Xinje XDPPro project, PLC1: XDH-60T4 (software 3.7.14b 2022-06-24)

PROGRAM 梯形图

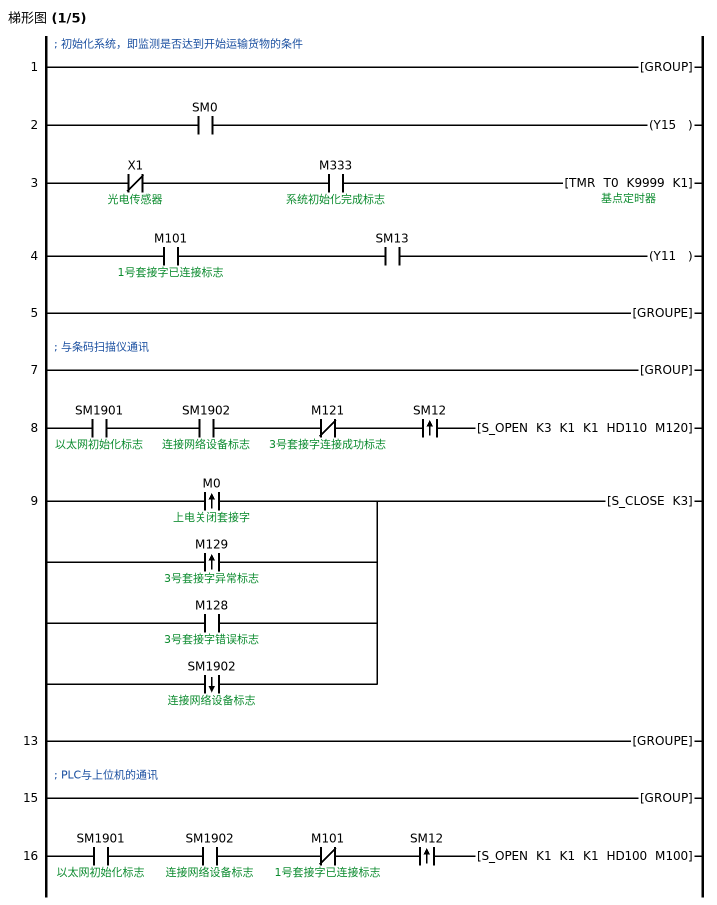
; 初始化系统，即监测是否达到开始运输货物的条件
GROUP
LD     SM0
OUT    Y15
LDI    X1	; 光电传感器
AND    M333	; 系统初始化完成标志
TMR    T0 K9999 K1	; 基点定时器
LD     M101	; 1号套接字已连接标志
AND    SM13
OUT    Y11
GROUPE
; 与条码扫描仪通讯
GROUP
LD     SM1901	; 以太网初始化标志
AND    SM1902	; 连接网络设备标志
ANI    M121	; 3号套接字连接成功标志
ANDP   SM12
S_OPEN K3 K1 K1 HD110 M120
LDP    M0	; 上电关闭套接字
ORP    M129	; 3号套接字异常标志
OR     M128	; 3号套接字错误标志
ORF    SM1902	; 连接网络设备标志
S_CLOSE K3
GROUPE
; PLC与上位机的通讯
GROUP
LD     SM1901	; 以太网初始化标志
AND    SM1902	; 连接网络设备标志
ANI    M101	; 1号套接字已连接标志
ANDP   SM12
S_OPEN K1 K1 K1 HD100 M100

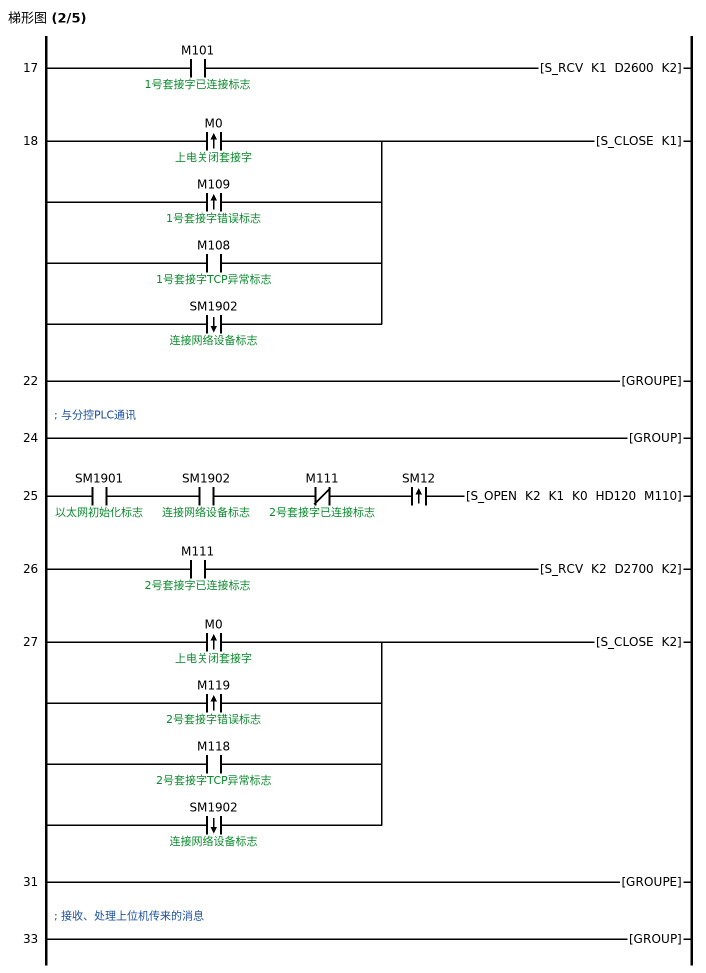
LD     M101	; 1号套接字已连接标志
S_RCV  K1 D2600 K2
LDP    M0	; 上电关闭套接字
ORP    M109	; 1号套接字错误标志
OR     M108	; 1号套接字TCP异常标志
ORF    SM1902	; 连接网络设备标志
S_CLOSE K1
GROUPE
; 与分控PLC通讯
GROUP
LD     SM1901	; 以太网初始化标志
AND    SM1902	; 连接网络设备标志
ANI    M111	; 2号套接字已连接标志
ANDP   SM12
S_OPEN K2 K1 K0 HD120 M110
LD     M111	; 2号套接字已连接标志
S_RCV  K2 D2700 K2
LDP    M0	; 上电关闭套接字
ORP    M119	; 2号套接字错误标志
OR     M118	; 2号套接字TCP异常标志
ORF    SM1902	; 连接网络设备标志
S_CLOSE K2
GROUPE
; 接收、处理上位机传来的消息
GROUP

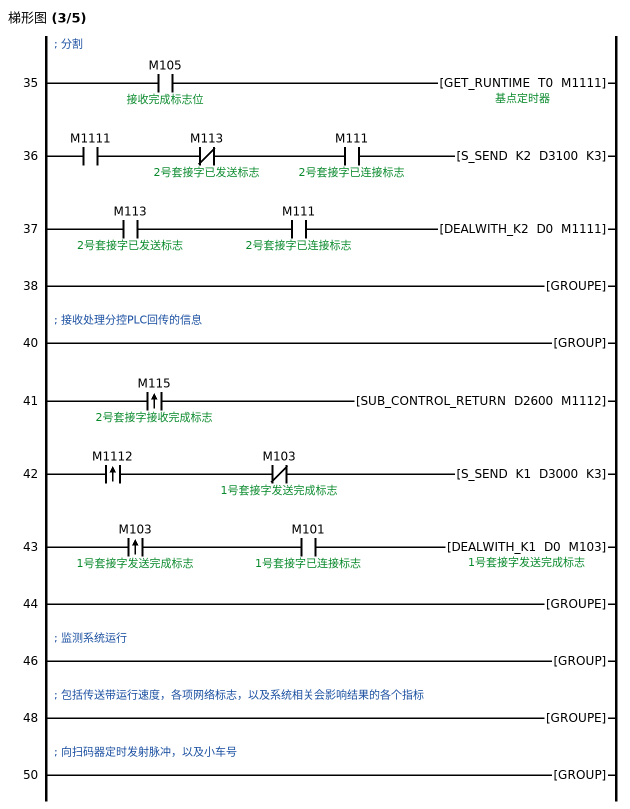
; 分割
LD     M105	; 接收完成标志位
GET_RUNTIME T0 M1111	; 基点定时器
LD     M1111
ANI    M113	; 2号套接字已发送标志
AND    M111	; 2号套接字已连接标志
S_SEND K2 D3100 K3
LD     M113	; 2号套接字已发送标志
AND    M111	; 2号套接字已连接标志
DEALWITH_K2 D0 M1111
GROUPE
; 接收处理分控PLC回传的信息
GROUP
LDP    M115	; 2号套接字接收完成标志
SUB_CONTROL_RETURN D2600 M1112
LDP    M1112
ANI    M103	; 1号套接字发送完成标志
S_SEND K1 D3000 K3
LDP    M103	; 1号套接字发送完成标志
AND    M101	; 1号套接字已连接标志
DEALWITH_K1 D0 M103	; 1号套接字发送完成标志
GROUPE
; 监测系统运行
GROUP
; 包括传送带运行速度，各项网络标志，以及系统相关会影响结果的各个指标
GROUPE
; 向扫码器定时发射脉冲，以及小车号
GROUP

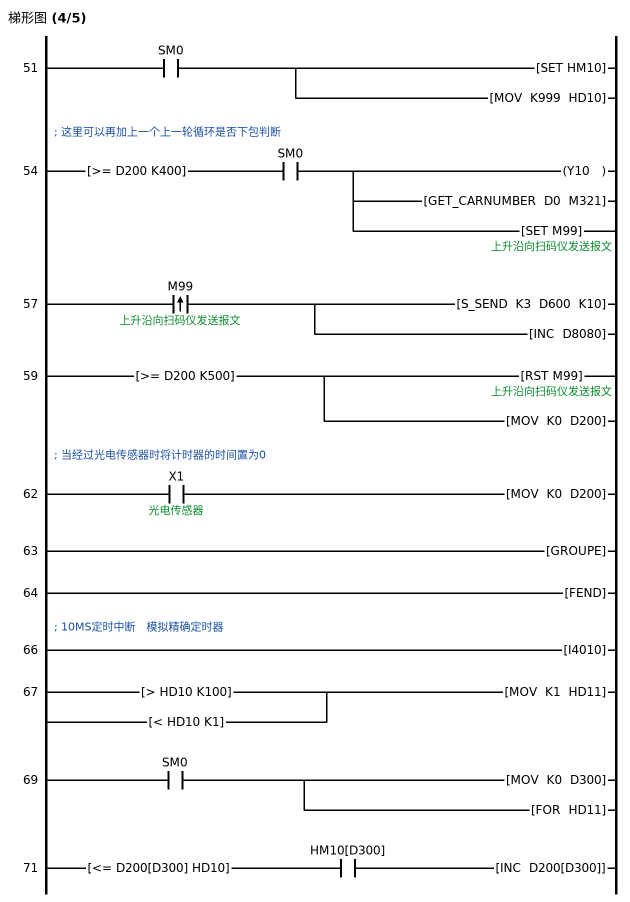
LD     SM0
SET    HM10
MOV    K999 HD10
; 这里可以再加上一个上一轮循环是否下包判断
LD>=   D200 K400
AND    SM0
OUT    Y10
GET_CARNUMBER D0 M321
SET    M99	; 上升沿向扫码仪发送报文
LDP    M99	; 上升沿向扫码仪发送报文
S_SEND K3 D600 K10
INC    D8080
LD>=   D200 K500
RST    M99	; 上升沿向扫码仪发送报文
MOV    K0 D200
; 当经过光电传感器时将计时器的时间置为0
LD     X1	; 光电传感器
MOV    K0 D200
GROUPE
FEND
; 10MS定时中断　模拟精确定时器
I4010
LD>    HD10 K100
OR<    HD10 K1
MOV    K1 HD11
LD     SM0
MOV    K0 D300
FOR    HD11
LD<=   D200[D300] HD10
AND    HM10[D300]
INC    D200[D300]

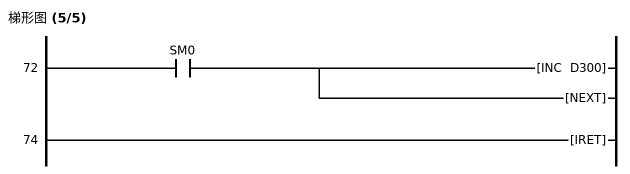
LD     SM0
INC    D300
NEXT
IRET

COMMENTS (devices not used above)
M1	1号套接字发送数据标志
HM0	手动建立连接
M2	1号套接字接收数据
M3	2号套接字发送数据标志
M4	2号套接字接收数据标志
Y6	给相机发脉冲
Y0	相机
Y7	接扫码仪

C FILE func1.h
#ifndef	_FUNC1_H
#define	_FUNC1_H
/*********宏定义用来存放需要的返回值************/
 #define NEEDTIME D[3100]       //保存返回值
 #define CAR      D[2600]        //存储判断出来的小车号
 #define Bourn     D[2605]       //目的格口
//#define Time      D[300]           //时间基点定时器的计数值 
#define D_D	     *(INT32S*)&D

/* 存放一些函数中需要的参数 
所有的距离单位为毫米，时间单位为毫秒
 */
 #define tmpp D_D[798]
 #define carnumber D_D[598]
 
 
INT32S TrackLength = 50000;           //轨道的长度
INT32S  Speed = 1;               //小车速度1mm/ms
INT32S DistanceOfCar = 400;      //小车的间距(单位为：毫米)
INT32S TIMELOSS = 5;          //电机启动时间偏移量(单位为：毫秒)

INT32S Time_Offset =0 ;           //时间偏移量，由于没有进行实验测试暂时设置为0,该值是用来计算小车上的电机转动所需要的时间

INT32S DistanceOfCut = 900;          //此处割口的间距 ————割口的长度加上割口间的距离

INT32S  Camera_Position = 600; //扫码设备的位置

INT32S Time = 0;               //距离时间基点的时间

INT32S Failure[20];

#endif

C FUNCTION BLOCK dealwith_k1.fcb
/* #EXPORT_ENTRY_BEGIN(DEALWITH_K1)
//    类型              模式             个数               映射          注释
W = { type = "PINT16S", mode = [In,Out], count = "unknown", map = [D,HD], comment = "" }
B = { type = "BIT"    , mode = [In,Out], count = "unknown", map = [M,HM], comment = "" }
#EXPORT_ENTRY_END */
/*************************************************************************
 * FunctionBlockName:  DEALWITH_K1
 * Version:            1.0.0
 * Author:             
 * UpdateTime:         2022-08-22 14:10:12
 * Comment:            
**************************************************************************/

/**
 * @summary 
 * @param W 
 * @param B 
 */
void DEALWITH_K1(PINT16S W,BIT B)
{
	#define SysRegAddr_HD_D_HM_M
    M[103] = 0;

}

C FUNCTION BLOCK dealwith_k2.fcb
/* #EXPORT_ENTRY_BEGIN(DEALWITH_K2)
//    类型              模式             个数               映射          注释
W = { type = "PINT16S", mode = [In,Out], count = "unknown", map = [D,HD], comment = "" }
B = { type = "BIT"    , mode = [In,Out], count = "unknown", map = [M,HM], comment = "" }
#EXPORT_ENTRY_END */
/*************************************************************************
 * FunctionBlockName:  DEALWITH_K2
 * Version:            1.0.0
 * Author:             
 * UpdateTime:         2022-08-22 14:08:06
 * Comment:            
**************************************************************************/

/**
 * @summary 
 * @param W 
 * @param B 
 */
void DEALWITH_K2(PINT16S W,BIT B)
{
	#define SysRegAddr_HD_D_HM_M
    M[113] = 0;
    M[1111] = 0;

}

C FUNCTION BLOCK func1.fcb
/* #EXPORT_ENTRY_BEGIN(FUNC1)
//    类型              模式             个数               映射          注释
W = { type = "PINT16S", mode = [In,Out], count = "unknown", map = [D,HD], comment = "" }
B = { type = "BIT"    , mode = [In,Out], count = "unknown", map = [M,HM], comment = "" }
#EXPORT_ENTRY_END */
/*************************************************************************
 * FunctionBlockName:  FUNC1
 * Version:            1.0.0
 * Author:             
 * UpdateTime:         2022-08-18 08:24:01
 * Comment:            
**************************************************************************/

/**
 * @summary 
 * @param W 
 * @param B 
 */
void FUNC1(PINT16S W,BIT B)
{
	#define SysRegAddr_HD_D_HM_M

}

C FUNCTION BLOCK get_carnumber.fcb
/* 输入时间，返回当前相机拍摄的小车号
#EXPORT_ENTRY_BEGIN(GET_CARNUMBER)
//    类型              模式             个数               映射          注释
W = { type = "PINT16S", mode = [In,Out], count = "unknown", map = [D,HD], comment = "" }
B = { type = "BIT"    , mode = [In,Out], count = "unknown", map = [M,HM], comment = "" }
#EXPORT_ENTRY_END */
/*************************************************************************
 * FunctionBlockName:  GET_CARNUMBER
 * Version:            1.0.0
 * Author:             rpl
 * UpdateTime:         2022-08-10 14:44:36
 * Comment:            输入时间，返回当前相机拍摄的小车号
**************************************************************************/

/**
 * @summary 
 * @param W 
 * @param B 
 */
 #include"func1.h"
 
 
void GET_CARNUMBER(PINT16S W,BIT B)
{
	#define SysRegAddr_HD_D_HM_M＿T
	/*根据时间判断出当前是多少号小车(小车从0号开始排序) */
     tmpp =  Speed * D[888] *10- Camera_Position;
    carnumber = ( tmpp / DistanceOfCar );  //判断是哪个小车，用来绑定小车的控制电机计时时间
    //CAR = 40;
    /***判断小车上的货物是否在上一轮没有卸载下来,暂不判断******/ 

    
    /***将小车号数据写入寄存器，起始位置Ｄ600,十个***/
        //消息头
    D[600] = 0x02;
    //功能位
    D[601] = 0x53;
    //千位
    D[602] = 0x30;
    
    //百位
    int ss= (D[598] /100) % 10；
    D[603] = 48+ss;
    
    //十位
    int  temp = 48 + (D[598] /10) % 10；
    D[604] = temp;
    
    //个位
    int  temp0 = 48 + D[598] % 10；
    D[605] = temp0;
    
    //结束符
    D[606] = 0x03;
    unsigned char LRC = 0;
    for(int i = 601;i<=605;i++)
    {
        LRC ^= D[i];
    }
    //LRC 校验
    D[607] = LRC;
    
    //尾字符
    D[608] = 0x0D;
    D[609] = 0x0A;
    
    
    
    M[321] = 1;
    return;
}

C FUNCTION BLOCK get_runtime.fcb
/* D[100]返回某个电机在多少秒后运行,D[101]返回判断出的小车号，以此来进行绑定
#EXPORT_ENTRY_BEGIN(GET_RUNTIME)
//    类型          模式             个数               映射          注释
w = { type = "BIT", mode = [In]    , count = "1"      , map = [T]   , comment = "时间差" }
B = { type = "BIT", mode = [In,Out], count = "unknown", map = [M,HM], comment = ""    }
#EXPORT_ENTRY_END */
/*************************************************************************
 * FunctionBlockName:  GET_RUNTIME
 * Version:            1.0.0
 * Author:             rpl
 * UpdateTime:         2022-07-25 16:38:06
 * Comment:            D[100]返回某个电机在多少秒后运行,D[101]返回判断出的小车号，以此来进行绑定
**************************************************************************/

/**
 * @summary 
 * @param w 时间差
 * @param B 
 */
 //#include "func1.h"

void GET_RUNTIME(BIT w,BIT B)
{
	#define SysRegAddr_HD_D_HM_M_T

    //Time = T[0] * 0.01;
    //if(Bourn * DistanceOfCut < Camera_Position ) //处理特殊情况：货物的目的地在光电传感器和拍照设备之间的情况
    //{
    	//NEEDTIME = (Bourn * DistanceOfCut + CAR * DistanceOfCar + TrackLength) / Speed   -  Time; 
    //} 
    //else{　//　正常情况
        
        //NEEDTIME = (Bourn * DistanceOfCut + CAR * DistanceOfCar) / Speed  - Time; //总时间减去已经用的时间
    //}
   // D[3101] = CAR;
    D[3102] = 121;
    M[105]  = 0;
    //D[2600] = 10;
    //D[2601] = 50;
    //Time = 200;
    //D[3101] = 151;
    //M[1111] = 1;
    
    
    
    
	
	
	
	
    //float sub = TrackLength - Number[0] * DistanceOfCar; //在光电传感器触发时该小车的位置m  
    ////float temp = ( sub + Speed * ( float ) Time );  //加上T时间内小车行走的距离
    //float current = temp > TrackLength ? temp - TrackLength : TrackLength - temp; //小车当前的位置
    
    //NEEDTIME = ( Bourn * DistanceOfCar - current ) / Speed  - Time_Offset; //路程除以速度得到时间
    //if(NEEDTIME<0) //处理在目的地在小车当前位置之前的情况
    //{
        //NEEDTIME = ( ( TrackLength - curren t ) + Bourn  * DistanceOfCar ) / Speed - Time_Offset;
    //}          
        
    return;
}

C FUNCTION BLOCK myt_rest.fcb
/* 将套接字的标志位全部复位
#EXPORT_ENTRY_BEGIN(MYT_REST)
//    类型          模式             个数               映射          注释
W = { type = "BIT", mode = [In,Out], count = "unknown", map = [M]   , comment = "" }
B = { type = "BIT", mode = [In,Out], count = "unknown", map = [M,HM], comment = "" }
#EXPORT_ENTRY_END */
/*************************************************************************
 * FunctionBlockName:  MYT_REST
 * Version:            1.0.0
 * Author:             rpl
 * UpdateTime:         2022-08-17 16:47:03
 * Comment:            将套接字的标志位全部复位
**************************************************************************/

/**
 * @summary 
 * @param W 
 * @param B 
 */
void MYT_REST(BIT W,BIT B)
{
	#define SysRegAddr_HD_D_HM_M
    //D[2600] = 0;
    //D[2601] = 0;
    //D[2602] = 0;
    //M[113] = 0;
}

C FUNCTION BLOCK process.fcb
/* 处理分控回传的数据
#EXPORT_ENTRY_BEGIN(PROCESS)
//    类型              模式             个数               映射          注释
W = { type = "PINT16S", mode = [In,Out], count = "unknown", map = [D,HD], comment = "" }
B = { type = "BIT"    , mode = [In,Out], count = "unknown", map = [M,HM], comment = "" }
#EXPORT_ENTRY_END */
/*************************************************************************
 * FunctionBlockName:  PROCESS
 * Version:            1.0.0
 * Author:             rpl
 * UpdateTime:         2022-08-18 10:58:38
 * Comment:            处理分控回传的数据
**************************************************************************/

/**
 * @summary 
 * @param W 
 * @param B 
 */
void PROCESS(PINT16S W,BIT B)
{
	#define SysRegAddr_HD_D_HM_M
	
	

}

C FUNCTION BLOCK setcamer.fcb
/* #EXPORT_ENTRY_BEGIN(SETCAMER)
//    类型              模式             个数               映射          注释
W = { type = "PINT16S", mode = [In,Out], count = "unknown", map = [D,HD], comment = "" }
B = { type = "BIT"    , mode = [In,Out], count = "unknown", map = [M,HM], comment = "" }
#EXPORT_ENTRY_END */
/*************************************************************************
 * FunctionBlockName:  SETCAMER
 * Version:            1.0.0
 * Author:             rpl
 * UpdateTime:         2022-08-25 16:03:02
 * Comment:            
**************************************************************************/

/**
 * @summary 
 * @param W 
 * @param B 
 */
void SETCAMER(PINT16S W,BIT B)
{
	#define SysRegAddr_HD_D_HM_M
    HM[10] = 1;

}

C FUNCTION BLOCK sub_control_return.fcb
/* 处理分控回传的数据
#EXPORT_ENTRY_BEGIN(SUB_CONTROL_RETURN)
//    类型              模式             个数               映射          注释
W = { type = "PINT16S", mode = [In,Out], count = "unknown", map = [D,HD], comment = "" }
B = { type = "BIT"    , mode = [In,Out], count = "unknown", map = [M,HM], comment = "" }
#EXPORT_ENTRY_END */
/*************************************************************************
 * FunctionBlockName:  SUB_CONTROL_RETURN
 * Version:            1.0.0
 * Author:             rpl
 * UpdateTime:         2022-08-19 10:53:12
 * Comment:            处理分控回传的数据
**************************************************************************/

/**
 * @summary 
 * @param W 
 * @param B 
 */
 
 
 /**分控plc回传的数据存放的首地址在D2700**/
 /**************
 D2700 唯一标识符
 D2701 小车号
 D2702 格口号
 D2703 投放成功或者失败
 
 ****************/
void SUB_CONTROL_RETURN(PINT16S W,BIT B)
{
    #define SysRegAddr_HD_D_HM_M
    /**如果投放失败则将该小车号存入未投放成功数组中**/
    //if ( D[2703] == 0 ) {
    //for ( int i = 0; i <= 20; i++ )
    //{
        //if ( Failure[i] == 0 )
            //Failure[i] = D[2701];
    //}
    D[3000] =  D[2700];
    D[3001] =  D[2701];
    D[3002] =  D[2702];
}